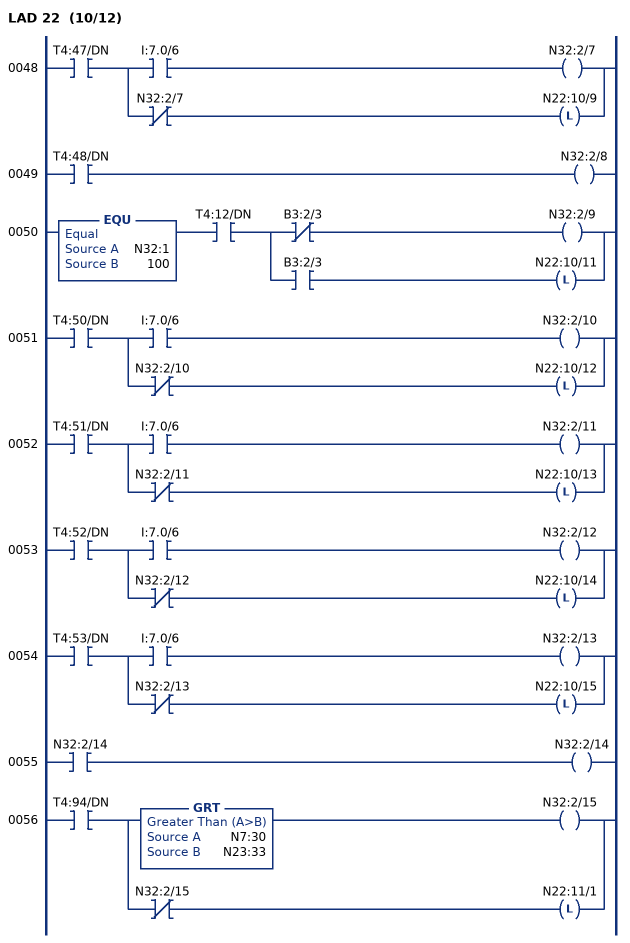
% Rung: 48 %
SOR XIC T4:47/DN BST XIC I:7.0/6 OTE N32:2/7 NXB XIO N32:2/7 OTL N22:10/9 BND EOR
% Rung: 49 %
SOR XIC T4:48/DN OTE N32:2/8 EOR
% Rung: 50 %
SOR EQU N32:1 100 XIC T4:12/DN BST XIO B3:2/3 OTE N32:2/9 NXB XIC B3:2/3 OTL N22:10/11 BND EOR
% Rung: 51 %
SOR XIC T4:50/DN BST XIC I:7.0/6 OTE N32:2/10 NXB XIO N32:2/10 OTL N22:10/12 BND EOR
% Rung: 52 %
SOR XIC T4:51/DN BST XIC I:7.0/6 OTE N32:2/11 NXB XIO N32:2/11 OTL N22:10/13 BND EOR
% Rung: 53 %
SOR XIC T4:52/DN BST XIC I:7.0/6 OTE N32:2/12 NXB XIO N32:2/12 OTL N22:10/14 BND EOR
% Rung: 54 %
SOR XIC T4:53/DN BST XIC I:7.0/6 OTE N32:2/13 NXB XIO N32:2/13 OTL N22:10/15 BND EOR
% Rung: 55 %
SOR XIC N32:2/14 OTE N32:2/14 EOR
% Rung: 56 %
SOR XIC T4:94/DN BST GRT N7:30 N23:33 OTE N32:2/15 NXB XIO N32:2/15 OTL N22:11/1 BND EOR

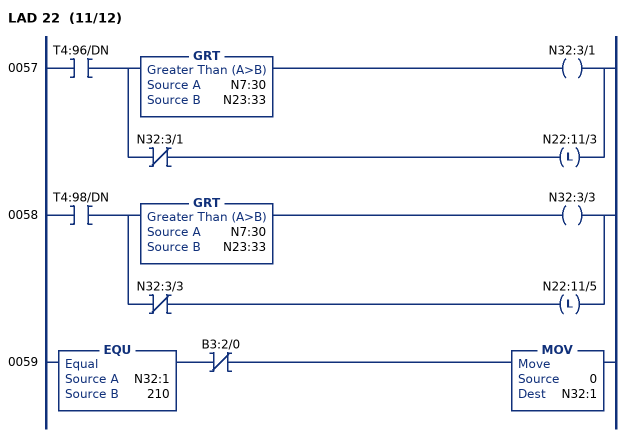
% Rung: 57 %
SOR XIC T4:96/DN BST GRT N7:30 N23:33 OTE N32:3/1 NXB XIO N32:3/1 OTL N22:11/3 BND EOR
% Rung: 58 %
SOR XIC T4:98/DN BST GRT N7:30 N23:33 OTE N32:3/3 NXB XIO N32:3/3 OTL N22:11/5 BND EOR
% Rung: 59 %
SOR EQU N32:1 210 XIO B3:2/0 MOV 0 N32:1 EOR

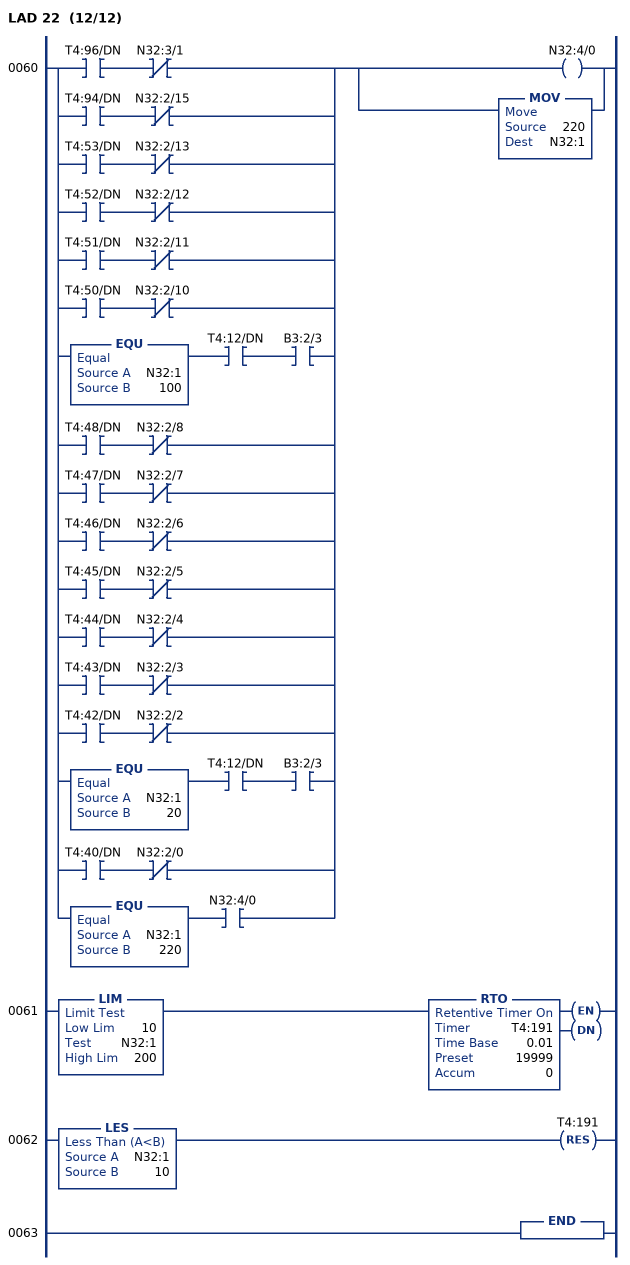
% Rung: 60 %
SOR BST XIC T4:96/DN XIO N32:3/1 NXB XIC T4:94/DN XIO N32:2/15 NXB XIC T4:53/DN XIO N32:2/13 NXB XIC T4:52/DN XIO N32:2/12 NXB XIC T4:51/DN XIO N32:2/11 NXB XIC T4:50/DN XIO N32:2/10 NXB EQU N32:1 100 XIC T4:12/DN XIC B3:2/3 NXB XIC T4:48/DN XIO N32:2/8 NXB XIC T4:47/DN XIO N32:2/7 NXB XIC T4:46/DN XIO N32:2/6 NXB XIC T4:45/DN XIO N32:2/5 NXB XIC T4:44/DN XIO N32:2/4 NXB XIC T4:43/DN XIO N32:2/3 NXB XIC T4:42/DN XIO N32:2/2 NXB EQU N32:1 20 XIC T4:12/DN XIC B3:2/3 NXB XIC T4:40/DN XIO N32:2/0 NXB EQU N32:1 220 XIC N32:4/0 BND BST OTE N32:4/0 NXB MOV 220 N32:1 BND EOR
% Rung: 61 %
SOR LIM 10 N32:1 200 RTO T4:191 0.01 19999 0 EOR
% Rung: 62 %
SOR LES N32:1 10 RES T4:191 EOR
% Rung: 63 %
SOR END EOR

LADDER 23
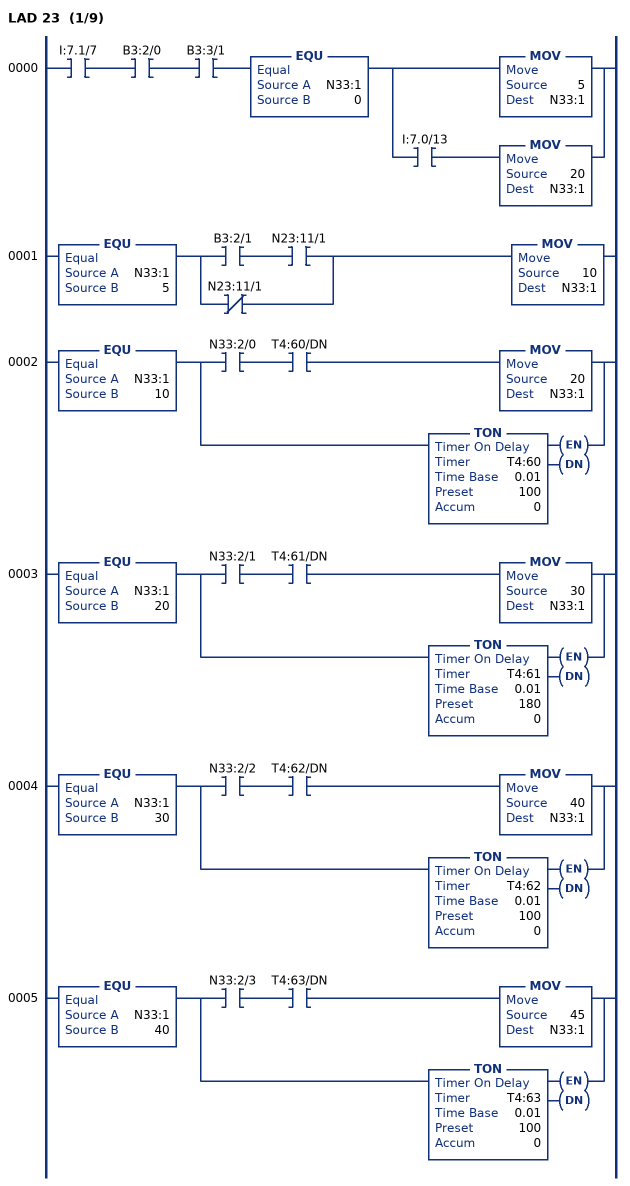
% Rung: 0 %
SOR XIC I:7.1/7 XIC B3:2/0 XIC B3:3/1 EQU N33:1 0 BST MOV 5 N33:1 NXB XIC I:7.0/13 MOV 20 N33:1 BND EOR
% Rung: 1 %
SOR EQU N33:1 5 BST XIC B3:2/1 XIC N23:11/1 NXB XIO N23:11/1 BND MOV 10 N33:1 EOR
% Rung: 2 %
SOR EQU N33:1 10 BST XIC N33:2/0 XIC T4:60/DN MOV 20 N33:1 NXB TON T4:60 0.01 100 0 BND EOR
% Rung: 3 %
SOR EQU N33:1 20 BST XIC N33:2/1 XIC T4:61/DN MOV 30 N33:1 NXB TON T4:61 0.01 180 0 BND EOR
% Rung: 4 %
SOR EQU N33:1 30 BST XIC N33:2/2 XIC T4:62/DN MOV 40 N33:1 NXB TON T4:62 0.01 100 0 BND EOR
% Rung: 5 %
SOR EQU N33:1 40 BST XIC N33:2/3 XIC T4:63/DN MOV 45 N33:1 NXB TON T4:63 0.01 100 0 BND EOR

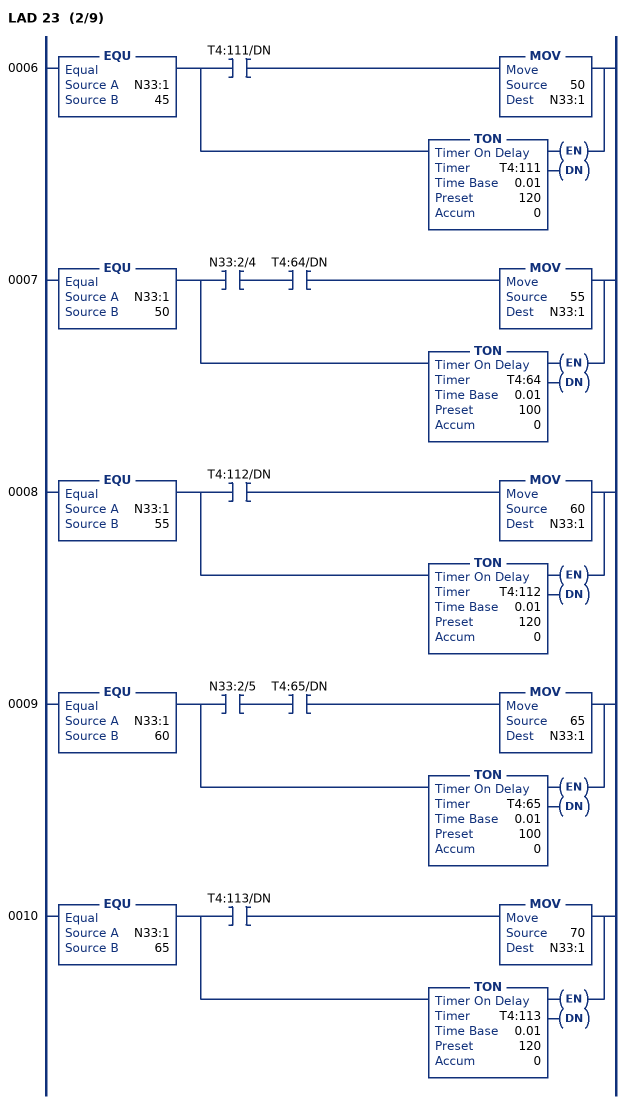
% Rung: 6 %
SOR EQU N33:1 45 BST XIC T4:111/DN MOV 50 N33:1 NXB TON T4:111 0.01 120 0 BND EOR
% Rung: 7 %
SOR EQU N33:1 50 BST XIC N33:2/4 XIC T4:64/DN MOV 55 N33:1 NXB TON T4:64 0.01 100 0 BND EOR
% Rung: 8 %
SOR EQU N33:1 55 BST XIC T4:112/DN MOV 60 N33:1 NXB TON T4:112 0.01 120 0 BND EOR
% Rung: 9 %
SOR EQU N33:1 60 BST XIC N33:2/5 XIC T4:65/DN MOV 65 N33:1 NXB TON T4:65 0.01 100 0 BND EOR
% Rung: 10 %
SOR EQU N33:1 65 BST XIC T4:113/DN MOV 70 N33:1 NXB TON T4:113 0.01 120 0 BND EOR

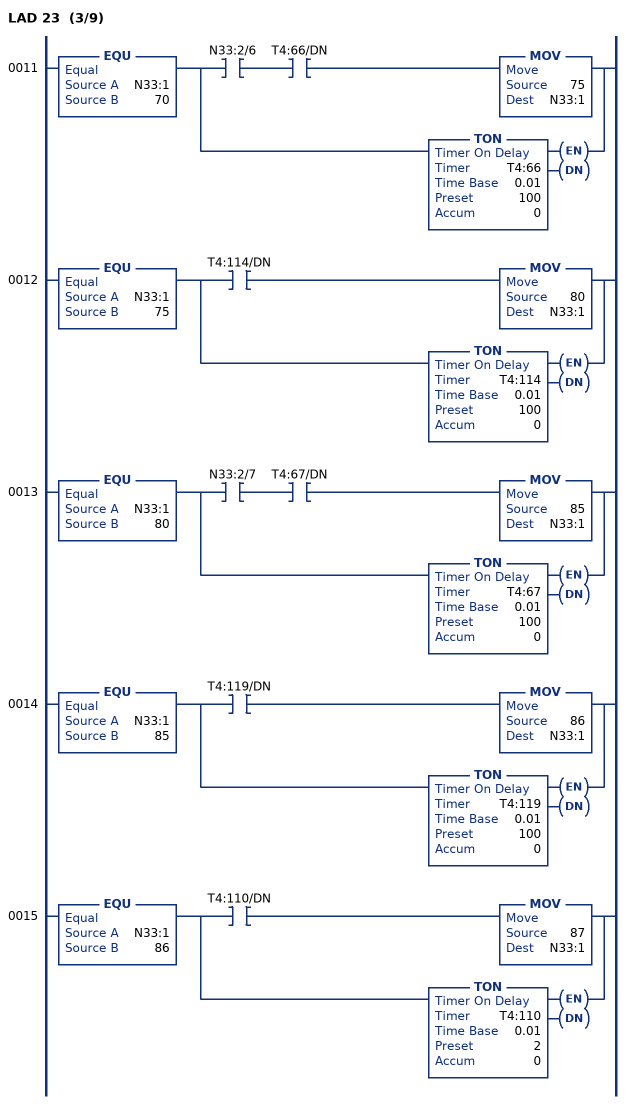
% Rung: 11 %
SOR EQU N33:1 70 BST XIC N33:2/6 XIC T4:66/DN MOV 75 N33:1 NXB TON T4:66 0.01 100 0 BND EOR
% Rung: 12 %
SOR EQU N33:1 75 BST XIC T4:114/DN MOV 80 N33:1 NXB TON T4:114 0.01 100 0 BND EOR
% Rung: 13 %
SOR EQU N33:1 80 BST XIC N33:2/7 XIC T4:67/DN MOV 85 N33:1 NXB TON T4:67 0.01 100 0 BND EOR
% Rung: 14 %
SOR EQU N33:1 85 BST XIC T4:119/DN MOV 86 N33:1 NXB TON T4:119 0.01 100 0 BND EOR
% Rung: 15 %
SOR EQU N33:1 86 BST XIC T4:110/DN MOV 87 N33:1 NXB TON T4:110 0.01 2 0 BND EOR

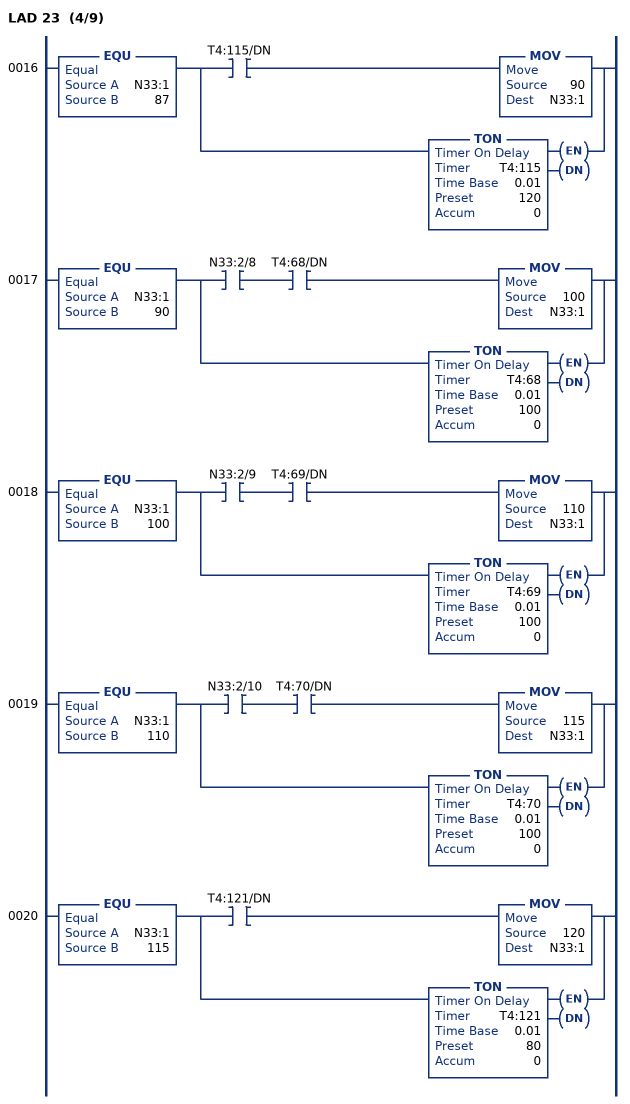
% Rung: 16 %
SOR EQU N33:1 87 BST XIC T4:115/DN MOV 90 N33:1 NXB TON T4:115 0.01 120 0 BND EOR
% Rung: 17 %
SOR EQU N33:1 90 BST XIC N33:2/8 XIC T4:68/DN MOV 100 N33:1 NXB TON T4:68 0.01 100 0 BND EOR
% Rung: 18 %
SOR EQU N33:1 100 BST XIC N33:2/9 XIC T4:69/DN MOV 110 N33:1 NXB TON T4:69 0.01 100 0 BND EOR
% Rung: 19 %
SOR EQU N33:1 110 BST XIC N33:2/10 XIC T4:70/DN MOV 115 N33:1 NXB TON T4:70 0.01 100 0 BND EOR
% Rung: 20 %
SOR EQU N33:1 115 BST XIC T4:121/DN MOV 120 N33:1 NXB TON T4:121 0.01 80 0 BND EOR

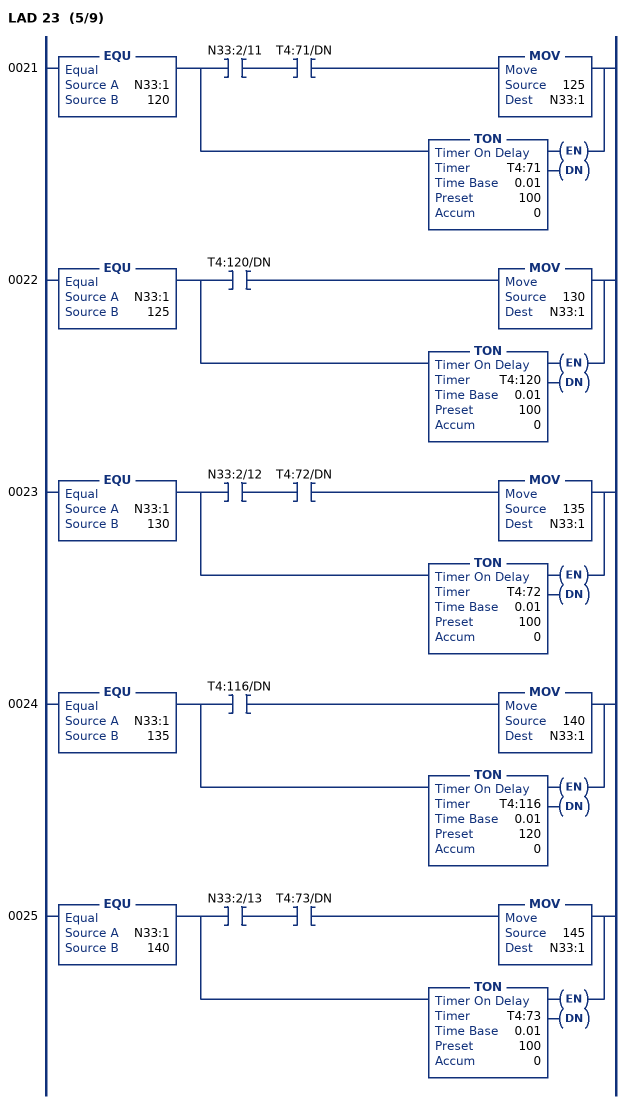
% Rung: 21 %
SOR EQU N33:1 120 BST XIC N33:2/11 XIC T4:71/DN MOV 125 N33:1 NXB TON T4:71 0.01 100 0 BND EOR
% Rung: 22 %
SOR EQU N33:1 125 BST XIC T4:120/DN MOV 130 N33:1 NXB TON T4:120 0.01 100 0 BND EOR
% Rung: 23 %
SOR EQU N33:1 130 BST XIC N33:2/12 XIC T4:72/DN MOV 135 N33:1 NXB TON T4:72 0.01 100 0 BND EOR
% Rung: 24 %
SOR EQU N33:1 135 BST XIC T4:116/DN MOV 140 N33:1 NXB TON T4:116 0.01 120 0 BND EOR
% Rung: 25 %
SOR EQU N33:1 140 BST XIC N33:2/13 XIC T4:73/DN MOV 145 N33:1 NXB TON T4:73 0.01 100 0 BND EOR

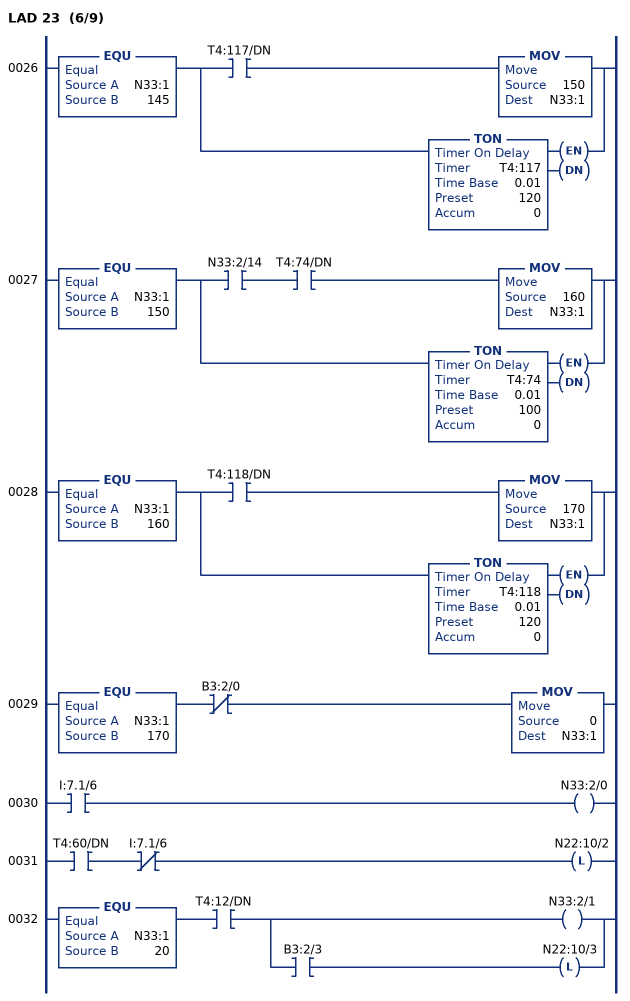
% Rung: 26 %
SOR EQU N33:1 145 BST XIC T4:117/DN MOV 150 N33:1 NXB TON T4:117 0.01 120 0 BND EOR
% Rung: 27 %
SOR EQU N33:1 150 BST XIC N33:2/14 XIC T4:74/DN MOV 160 N33:1 NXB TON T4:74 0.01 100 0 BND EOR
% Rung: 28 %
SOR EQU N33:1 160 BST XIC T4:118/DN MOV 170 N33:1 NXB TON T4:118 0.01 120 0 BND EOR
% Rung: 29 %
SOR EQU N33:1 170 XIO B3:2/0 MOV 0 N33:1 EOR
% Rung: 30 %
SOR XIC I:7.1/6 OTE N33:2/0 EOR
% Rung: 31 %
SOR XIC T4:60/DN XIO I:7.1/6 OTL N22:10/2 EOR
% Rung: 32 %
SOR EQU N33:1 20 XIC T4:12/DN BST OTE N33:2/1 NXB XIC B3:2/3 OTL N22:10/3 BND EOR

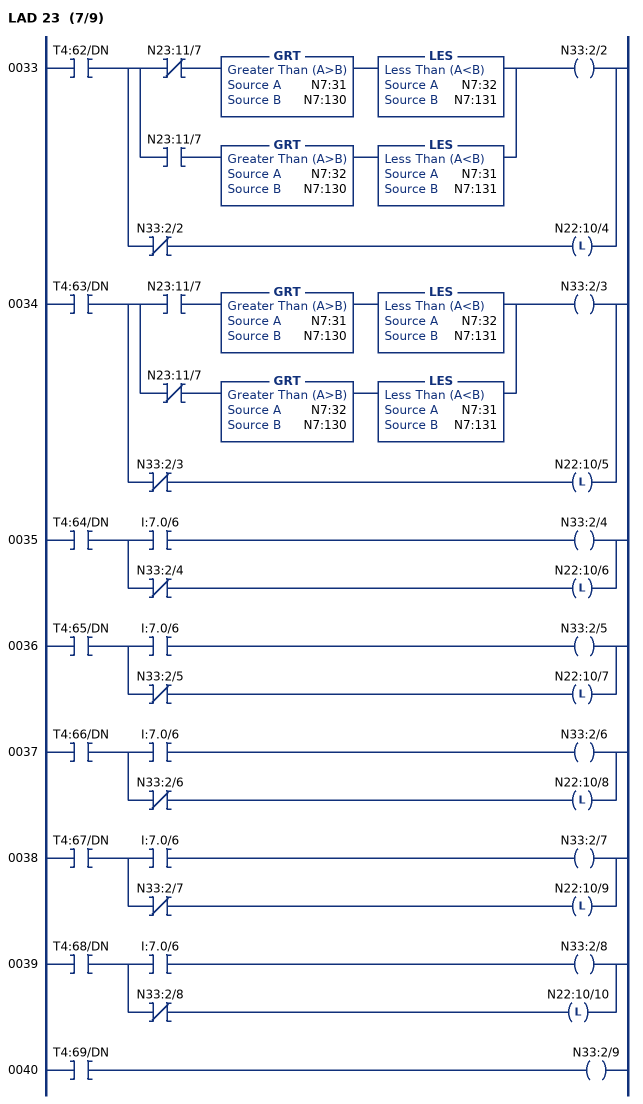
% Rung: 33 %
SOR XIC T4:62/DN BST BST XIO N23:11/7 GRT N7:31 N7:130 LES N7:32 N7:131 NXB XIC N23:11/7 GRT N7:32 N7:130 LES N7:31 N7:131 BND OTE N33:2/2 NXB XIO N33:2/2 OTL N22:10/4 BND EOR
% Rung: 34 %
SOR XIC T4:63/DN BST BST XIC N23:11/7 GRT N7:31 N7:130 LES N7:32 N7:131 NXB XIO N23:11/7 GRT N7:32 N7:130 LES N7:31 N7:131 BND OTE N33:2/3 NXB XIO N33:2/3 OTL N22:10/5 BND EOR
% Rung: 35 %
SOR XIC T4:64/DN BST XIC I:7.0/6 OTE N33:2/4 NXB XIO N33:2/4 OTL N22:10/6 BND EOR
% Rung: 36 %
SOR XIC T4:65/DN BST XIC I:7.0/6 OTE N33:2/5 NXB XIO N33:2/5 OTL N22:10/7 BND EOR
% Rung: 37 %
SOR XIC T4:66/DN BST XIC I:7.0/6 OTE N33:2/6 NXB XIO N33:2/6 OTL N22:10/8 BND EOR
% Rung: 38 %
SOR XIC T4:67/DN BST XIC I:7.0/6 OTE N33:2/7 NXB XIO N33:2/7 OTL N22:10/9 BND EOR
% Rung: 39 %
SOR XIC T4:68/DN BST XIC I:7.0/6 OTE N33:2/8 NXB XIO N33:2/8 OTL N22:10/10 BND EOR
% Rung: 40 %
SOR XIC T4:69/DN OTE N33:2/9 EOR

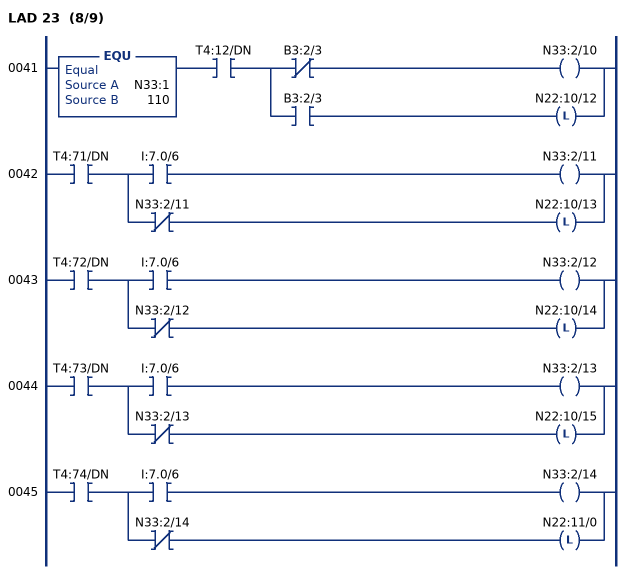
% Rung: 41 %
SOR EQU N33:1 110 XIC T4:12/DN BST XIO B3:2/3 OTE N33:2/10 NXB XIC B3:2/3 OTL N22:10/12 BND EOR
% Rung: 42 %
SOR XIC T4:71/DN BST XIC I:7.0/6 OTE N33:2/11 NXB XIO N33:2/11 OTL N22:10/13 BND EOR
% Rung: 43 %
SOR XIC T4:72/DN BST XIC I:7.0/6 OTE N33:2/12 NXB XIO N33:2/12 OTL N22:10/14 BND EOR
% Rung: 44 %
SOR XIC T4:73/DN BST XIC I:7.0/6 OTE N33:2/13 NXB XIO N33:2/13 OTL N22:10/15 BND EOR
% Rung: 45 %
SOR XIC T4:74/DN BST XIC I:7.0/6 OTE N33:2/14 NXB XIO N33:2/14 OTL N22:11/0 BND EOR

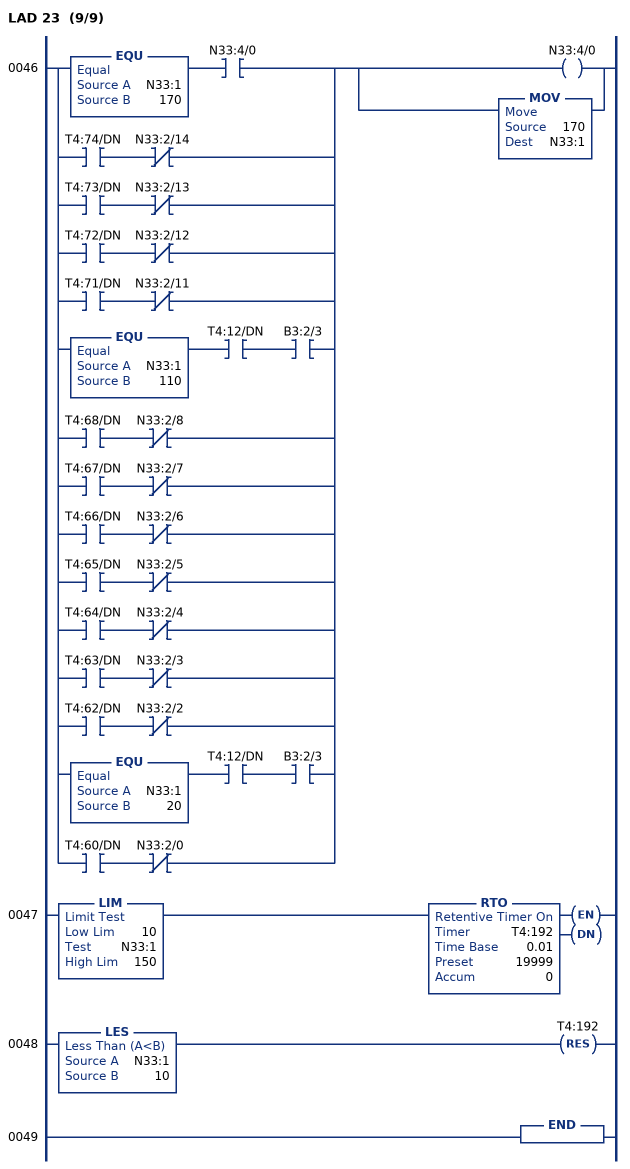
% Rung: 46 %
SOR BST EQU N33:1 170 XIC N33:4/0 NXB XIC T4:74/DN XIO N33:2/14 NXB XIC T4:73/DN XIO N33:2/13 NXB XIC T4:72/DN XIO N33:2/12 NXB XIC T4:71/DN XIO N33:2/11 NXB EQU N33:1 110 XIC T4:12/DN XIC B3:2/3 NXB XIC T4:68/DN XIO N33:2/8 NXB XIC T4:67/DN XIO N33:2/7 NXB XIC T4:66/DN XIO N33:2/6 NXB XIC T4:65/DN XIO N33:2/5 NXB XIC T4:64/DN XIO N33:2/4 NXB XIC T4:63/DN XIO N33:2/3 NXB XIC T4:62/DN XIO N33:2/2 NXB EQU N33:1 20 XIC T4:12/DN XIC B3:2/3 NXB XIC T4:60/DN XIO N33:2/0 BND BST OTE N33:4/0 NXB MOV 170 N33:1 BND EOR
% Rung: 47 %
SOR LIM 10 N33:1 150 RTO T4:192 0.01 19999 0 EOR
% Rung: 48 %
SOR LES N33:1 10 RES T4:192 EOR
% Rung: 49 %
SOR END EOR

LADDER 24
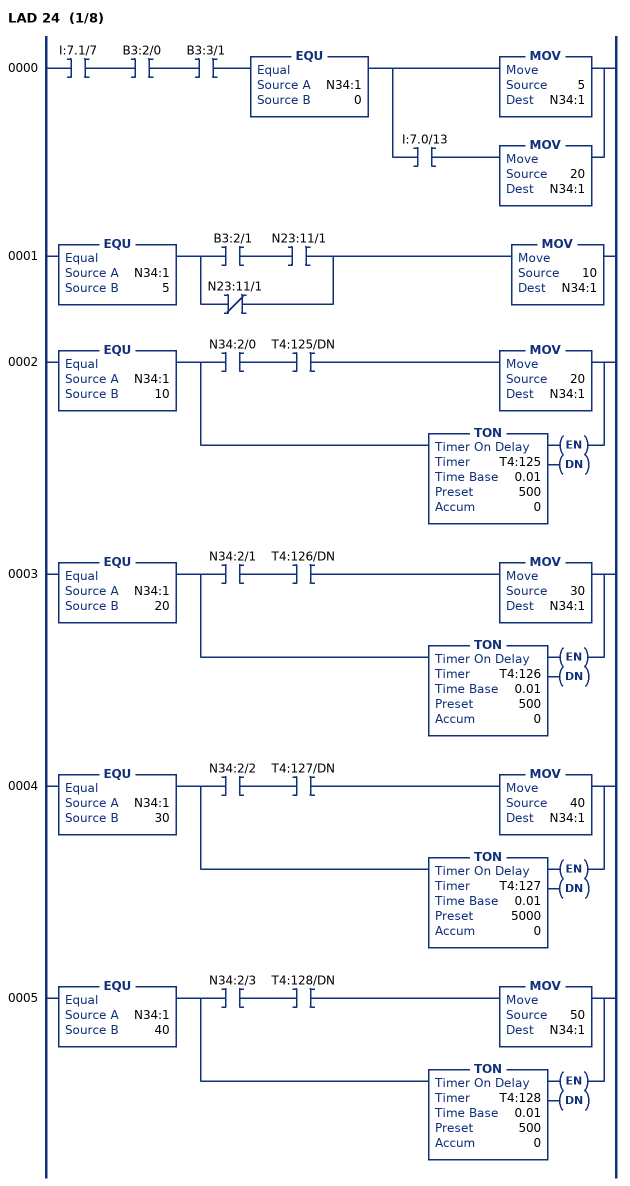
% Rung: 0 %
SOR XIC I:7.1/7 XIC B3:2/0 XIC B3:3/1 EQU N34:1 0 BST MOV 5 N34:1 NXB XIC I:7.0/13 MOV 20 N34:1 BND EOR
% Rung: 1 %
SOR EQU N34:1 5 BST XIC B3:2/1 XIC N23:11/1 NXB XIO N23:11/1 BND MOV 10 N34:1 EOR
% Rung: 2 %
SOR EQU N34:1 10 BST XIC N34:2/0 XIC T4:125/DN MOV 20 N34:1 NXB TON T4:125 0.01 500 0 BND EOR
% Rung: 3 %
SOR EQU N34:1 20 BST XIC N34:2/1 XIC T4:126/DN MOV 30 N34:1 NXB TON T4:126 0.01 500 0 BND EOR
% Rung: 4 %
SOR EQU N34:1 30 BST XIC N34:2/2 XIC T4:127/DN MOV 40 N34:1 NXB TON T4:127 0.01 5000 0 BND EOR
% Rung: 5 %
SOR EQU N34:1 40 BST XIC N34:2/3 XIC T4:128/DN MOV 50 N34:1 NXB TON T4:128 0.01 500 0 BND EOR

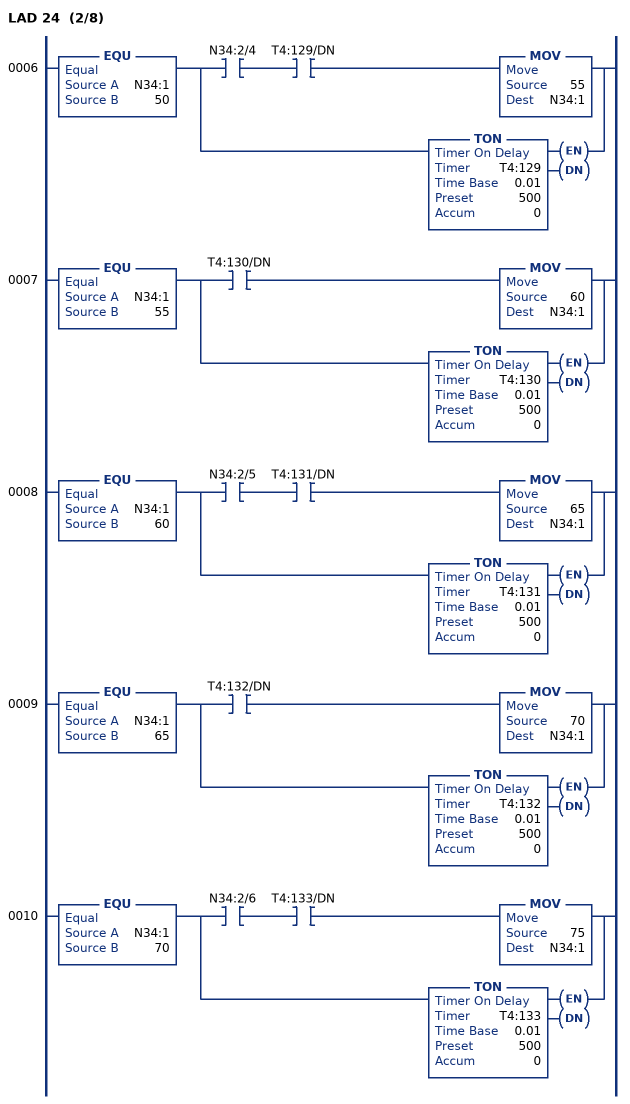
% Rung: 6 %
SOR EQU N34:1 50 BST XIC N34:2/4 XIC T4:129/DN MOV 55 N34:1 NXB TON T4:129 0.01 500 0 BND EOR
% Rung: 7 %
SOR EQU N34:1 55 BST XIC T4:130/DN MOV 60 N34:1 NXB TON T4:130 0.01 500 0 BND EOR
% Rung: 8 %
SOR EQU N34:1 60 BST XIC N34:2/5 XIC T4:131/DN MOV 65 N34:1 NXB TON T4:131 0.01 500 0 BND EOR
% Rung: 9 %
SOR EQU N34:1 65 BST XIC T4:132/DN MOV 70 N34:1 NXB TON T4:132 0.01 500 0 BND EOR
% Rung: 10 %
SOR EQU N34:1 70 BST XIC N34:2/6 XIC T4:133/DN MOV 75 N34:1 NXB TON T4:133 0.01 500 0 BND EOR

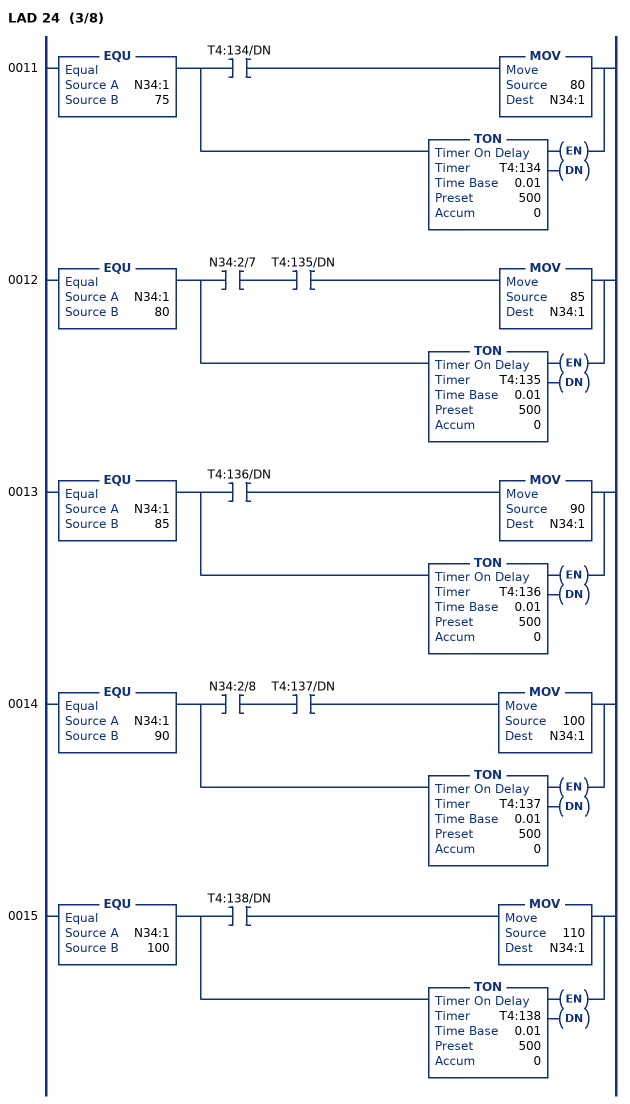
% Rung: 11 %
SOR EQU N34:1 75 BST XIC T4:134/DN MOV 80 N34:1 NXB TON T4:134 0.01 500 0 BND EOR
% Rung: 12 %
SOR EQU N34:1 80 BST XIC N34:2/7 XIC T4:135/DN MOV 85 N34:1 NXB TON T4:135 0.01 500 0 BND EOR
% Rung: 13 %
SOR EQU N34:1 85 BST XIC T4:136/DN MOV 90 N34:1 NXB TON T4:136 0.01 500 0 BND EOR
% Rung: 14 %
SOR EQU N34:1 90 BST XIC N34:2/8 XIC T4:137/DN MOV 100 N34:1 NXB TON T4:137 0.01 500 0 BND EOR
% Rung: 15 %
SOR EQU N34:1 100 BST XIC T4:138/DN MOV 110 N34:1 NXB TON T4:138 0.01 500 0 BND EOR

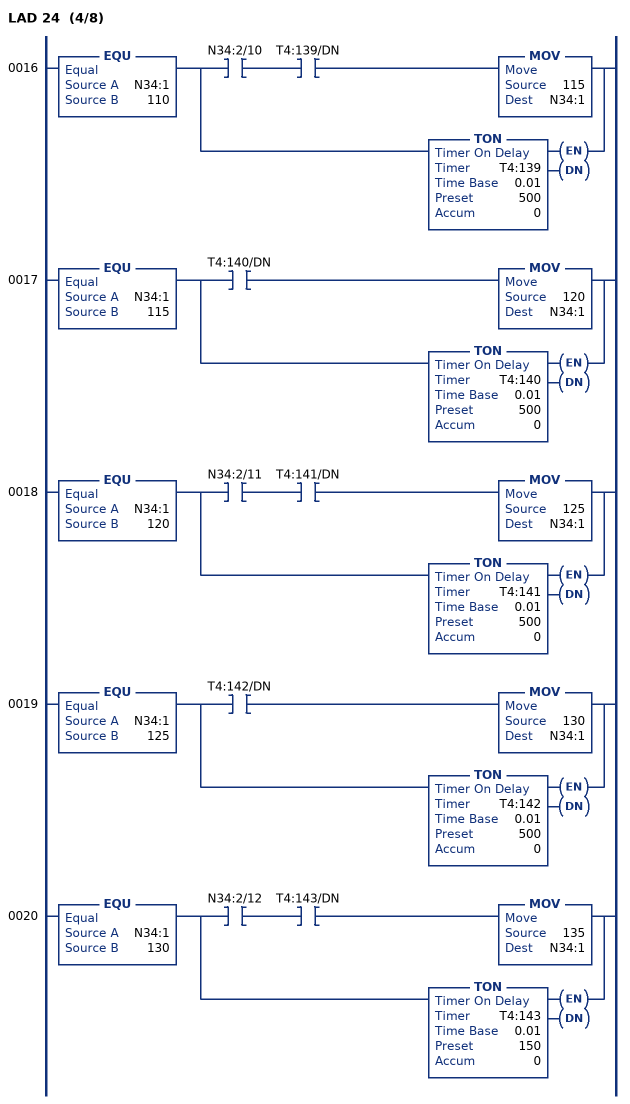
% Rung: 16 %
SOR EQU N34:1 110 BST XIC N34:2/10 XIC T4:139/DN MOV 115 N34:1 NXB TON T4:139 0.01 500 0 BND EOR
% Rung: 17 %
SOR EQU N34:1 115 BST XIC T4:140/DN MOV 120 N34:1 NXB TON T4:140 0.01 500 0 BND EOR
% Rung: 18 %
SOR EQU N34:1 120 BST XIC N34:2/11 XIC T4:141/DN MOV 125 N34:1 NXB TON T4:141 0.01 500 0 BND EOR
% Rung: 19 %
SOR EQU N34:1 125 BST XIC T4:142/DN MOV 130 N34:1 NXB TON T4:142 0.01 500 0 BND EOR
% Rung: 20 %
SOR EQU N34:1 130 BST XIC N34:2/12 XIC T4:143/DN MOV 135 N34:1 NXB TON T4:143 0.01 150 0 BND EOR

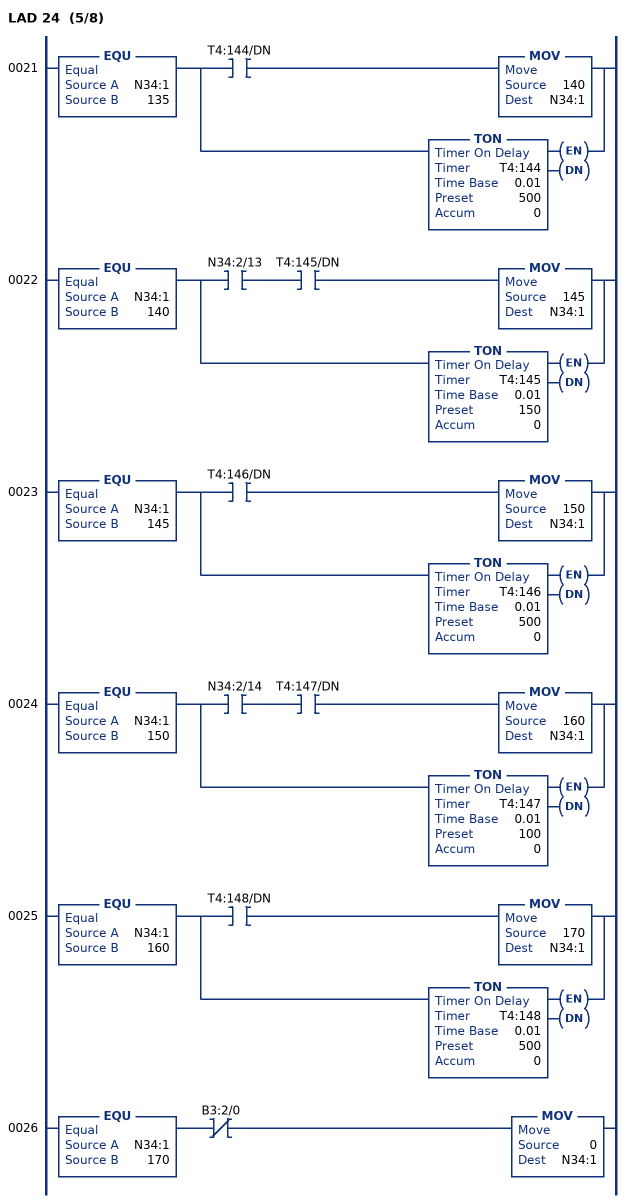
% Rung: 21 %
SOR EQU N34:1 135 BST XIC T4:144/DN MOV 140 N34:1 NXB TON T4:144 0.01 500 0 BND EOR
% Rung: 22 %
SOR EQU N34:1 140 BST XIC N34:2/13 XIC T4:145/DN MOV 145 N34:1 NXB TON T4:145 0.01 150 0 BND EOR
% Rung: 23 %
SOR EQU N34:1 145 BST XIC T4:146/DN MOV 150 N34:1 NXB TON T4:146 0.01 500 0 BND EOR
% Rung: 24 %
SOR EQU N34:1 150 BST XIC N34:2/14 XIC T4:147/DN MOV 160 N34:1 NXB TON T4:147 0.01 100 0 BND EOR
% Rung: 25 %
SOR EQU N34:1 160 BST XIC T4:148/DN MOV 170 N34:1 NXB TON T4:148 0.01 500 0 BND EOR
% Rung: 26 %
SOR EQU N34:1 170 XIO B3:2/0 MOV 0 N34:1 EOR

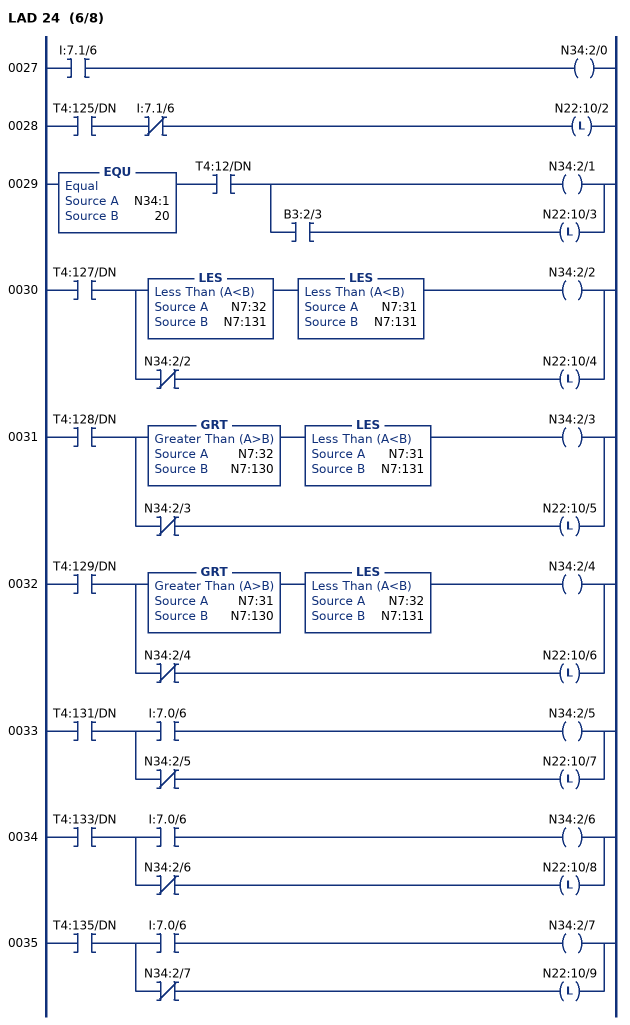
% Rung: 27 %
SOR XIC I:7.1/6 OTE N34:2/0 EOR
% Rung: 28 %
SOR XIC T4:125/DN XIO I:7.1/6 OTL N22:10/2 EOR
% Rung: 29 %
SOR EQU N34:1 20 XIC T4:12/DN BST OTE N34:2/1 NXB XIC B3:2/3 OTL N22:10/3 BND EOR
% Rung: 30 %
SOR XIC T4:127/DN BST LES N7:32 N7:131 LES N7:31 N7:131 OTE N34:2/2 NXB XIO N34:2/2 OTL N22:10/4 BND EOR
% Rung: 31 %
SOR XIC T4:128/DN BST GRT N7:32 N7:130 LES N7:31 N7:131 OTE N34:2/3 NXB XIO N34:2/3 OTL N22:10/5 BND EOR
% Rung: 32 %
SOR XIC T4:129/DN BST GRT N7:31 N7:130 LES N7:32 N7:131 OTE N34:2/4 NXB XIO N34:2/4 OTL N22:10/6 BND EOR
% Rung: 33 %
SOR XIC T4:131/DN BST XIC I:7.0/6 OTE N34:2/5 NXB XIO N34:2/5 OTL N22:10/7 BND EOR
% Rung: 34 %
SOR XIC T4:133/DN BST XIC I:7.0/6 OTE N34:2/6 NXB XIO N34:2/6 OTL N22:10/8 BND EOR
% Rung: 35 %
SOR XIC T4:135/DN BST XIC I:7.0/6 OTE N34:2/7 NXB XIO N34:2/7 OTL N22:10/9 BND EOR

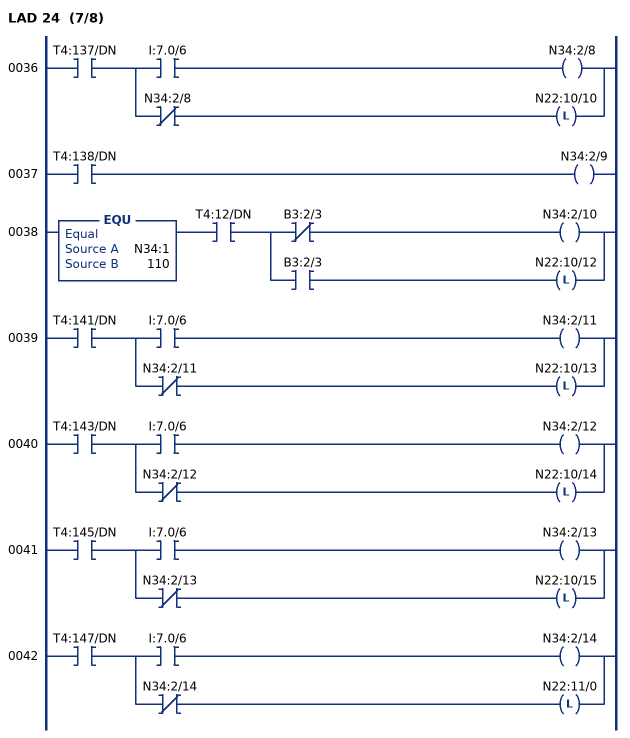
% Rung: 36 %
SOR XIC T4:137/DN BST XIC I:7.0/6 OTE N34:2/8 NXB XIO N34:2/8 OTL N22:10/10 BND EOR
% Rung: 37 %
SOR XIC T4:138/DN OTE N34:2/9 EOR
% Rung: 38 %
SOR EQU N34:1 110 XIC T4:12/DN BST XIO B3:2/3 OTE N34:2/10 NXB XIC B3:2/3 OTL N22:10/12 BND EOR
% Rung: 39 %
SOR XIC T4:141/DN BST XIC I:7.0/6 OTE N34:2/11 NXB XIO N34:2/11 OTL N22:10/13 BND EOR
% Rung: 40 %
SOR XIC T4:143/DN BST XIC I:7.0/6 OTE N34:2/12 NXB XIO N34:2/12 OTL N22:10/14 BND EOR
% Rung: 41 %
SOR XIC T4:145/DN BST XIC I:7.0/6 OTE N34:2/13 NXB XIO N34:2/13 OTL N22:10/15 BND EOR
% Rung: 42 %
SOR XIC T4:147/DN BST XIC I:7.0/6 OTE N34:2/14 NXB XIO N34:2/14 OTL N22:11/0 BND EOR

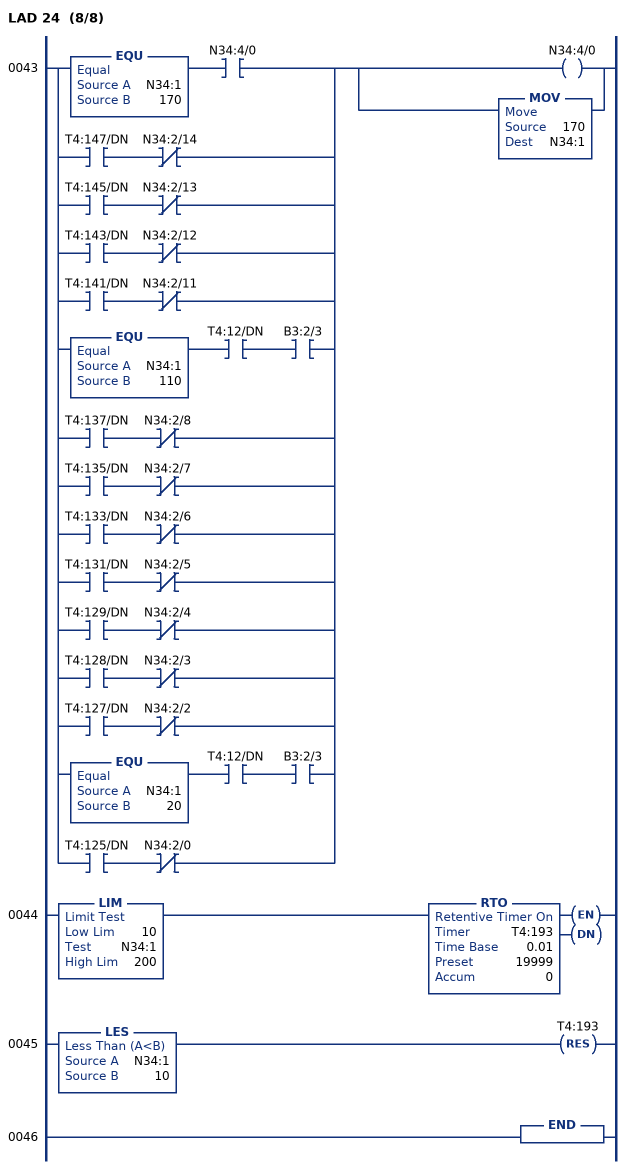
% Rung: 43 %
SOR BST EQU N34:1 170 XIC N34:4/0 NXB XIC T4:147/DN XIO N34:2/14 NXB XIC T4:145/DN XIO N34:2/13 NXB XIC T4:143/DN XIO N34:2/12 NXB XIC T4:141/DN XIO N34:2/11 NXB EQU N34:1 110 XIC T4:12/DN XIC B3:2/3 NXB XIC T4:137/DN XIO N34:2/8 NXB XIC T4:135/DN XIO N34:2/7 NXB XIC T4:133/DN XIO N34:2/6 NXB XIC T4:131/DN XIO N34:2/5 NXB XIC T4:129/DN XIO N34:2/4 NXB XIC T4:128/DN XIO N34:2/3 NXB XIC T4:127/DN XIO N34:2/2 NXB EQU N34:1 20 XIC T4:12/DN XIC B3:2/3 NXB XIC T4:125/DN XIO N34:2/0 BND BST OTE N34:4/0 NXB MOV 170 N34:1 BND EOR
% Rung: 44 %
SOR LIM 10 N34:1 200 RTO T4:193 0.01 19999 0 EOR
% Rung: 45 %
SOR LES N34:1 10 RES T4:193 EOR
% Rung: 46 %
SOR END EOR

DATA TABLE (non-zero values as saved)
DATA B3
% B3:0 % 0X8003 0X0005 0X0002 0X0001 0X0000 0X0000 0X0000 0X0000 0X0000 0X0000
DATA T4
% .PRE .ACC %
% T4:0 % 3 1
% T4:1 % 2 0
% T4:2 % 10 0
% T4:3 % 2 0
% T4:4 % 50 0
% T4:5 % 50 0
% T4:6 % 2 2
% T4:7 % 1 1
% T4:8 % 20 20
% T4:9 % 100 100
% T4:10 % 50 0
% T4:11 % 50 0
% T4:12 % 150 0
% T4:13 % 167 0
% T4:14 % 166 0
% T4:15 % 50 50
% T4:16 % 60 0
% T4:17 % 90 0
% T4:18 % 170 0
% T4:19 % 30 30
% T4:20 % 100 0
% T4:21 % 100 0
% T4:22 % 50 0
% T4:23 % 100 0
% T4:24 % 150 0
% T4:25 % 150 0
% T4:26 % 100 0
% T4:27 % 150 0
% T4:28 % 30 0
% T4:29 % 100 0
% T4:30 % 150 0
% T4:31 % 150 0
% T4:32 % 100 0
% T4:33 % 350 0
% T4:34 % 100 0
% T4:35 % 350 0
% T4:36 % 150 0
% T4:37 % 150 0
% T4:38 % 100 0
% T4:39 % 50 0
% T4:40 % 100 0
% T4:41 % 20 0
% T4:42 % 90 0
% T4:43 % 90 0
% T4:44 % 150 0
% T4:45 % 150 0
% T4:46 % 150 0
% T4:47 % 150 0
% T4:48 % 20 0
% T4:49 % 70 0
% T4:50 % 150 0
% T4:51 % 150 0
% T4:52 % 150 0
% T4:53 % 150 0
% T4:54 % 100 0
% T4:55 % 10 0
% T4:56 % 70 0
% T4:57 % 70 0
% T4:58 % 110 0
% T4:59 % 110 0
% T4:60 % 100 0
% T4:61 % 180 0
% T4:62 % 100 0
% T4:63 % 100 0
% T4:64 % 100 0
% T4:65 % 100 0
% T4:66 % 100 0
% T4:67 % 100 0
% T4:68 % 100 0
% T4:69 % 100 0
% T4:70 % 100 0
% T4:71 % 100 0
% T4:72 % 100 0
% T4:73 % 100 0
% T4:74 % 100 0
% T4:75 % 100 0
% T4:76 % 200 0
% T4:77 % 100 0
% T4:78 % 50 0
% T4:80 % 60 0
% T4:81 % 60 0
% T4:82 % 60 0
% T4:83 % 60 0
% T4:84 % 60 0
% T4:85 % 60 0
% T4:86 % 60 0
% T4:87 % 60 0
% T4:88 % 60 0
% T4:89 % 100 0
% T4:90 % 80 0
% T4:91 % 50 0
% T4:92 % 50 0
% T4:93 % 100 0
% T4:94 % 500 0
% T4:95 % 500 0
% T4:96 % 500 0
% T4:97 % 600 0
% T4:98 % 500 0
% T4:99 % 200 0
% T4:100 % 200 0
% T4:101 % 200 0
% T4:102 % 200 0
% T4:103 % 100 0
% T4:104 % 100 0
% T4:105 % 120 0
% T4:106 % 120 0
% T4:107 % 120 0
% T4:108 % 120 0
% T4:109 % 120 0
% T4:110 % 2 0
% T4:111 % 120 0
% T4:112 % 120 0
% T4:113 % 120 0
% T4:114 % 100 0
% T4:115 % 120 0
% T4:116 % 120 0
% T4:117 % 120 0
% T4:118 % 120 0
% T4:119 % 100 0
% T4:120 % 100 0
% T4:121 % 80 0
% T4:125 % 500 0
% T4:126 % 500 0
% T4:127 % 5000 0
% T4:128 % 500 0
% T4:129 % 500 0
% T4:130 % 500 0
% T4:131 % 500 0
% T4:132 % 500 0
% T4:133 % 500 0
% T4:134 % 500 0
% T4:135 % 500 0
% T4:136 % 500 0
% T4:137 % 500 0
% T4:138 % 500 0
% T4:139 % 500 0
% T4:140 % 500 0
% T4:141 % 500 0
% T4:142 % 500 0
% T4:143 % 150 0
% T4:144 % 500 0
% T4:145 % 150 0
% T4:146 % 500 0
% T4:147 % 100 0
% T4:148 % 500 0
% T4:190 % 19999 0
% T4:191 % 19999 0
% T4:192 % 19999 0
% T4:193 % 19999 0
% T4:199 % 150 0
DATA N7
% N7:0 % 30 102 0 0 200 400 1870 0 0 0
% N7:10 % 30 102 0 0 200 400 1870 0 0 0
% N7:20 % 0 76 0 0 0 0 0 1870 102 30
% N7:30 % -50 -25 -25 0 0 0 0 0 0 0
% N7:50 % 0 1 1 0 0 0 0 0 0 0
% N7:60 % 10 2 102 0 0 0 0 0 0 0
% N7:80 % 2 75 150 5 167 333 0 0 0 0
% N7:90 % 0 0 0 0 0 0 0 0 1 3
% N7:100 % 1 0 0 80 0 0 0 0 0 0
% N7:110 % 20 20 15 0 0 82 10 0 0 0
% N7:130 % 68 12 0 0 0 0 0 0 0 0
DATA F8
% F8:0 % 0 102 1 0 0
% F8:5 % 0.85 0.15 0.5 0.5 3
DATA ST20
% ST20:0 % ".01\0A\0D"
% ST20:1 % "1"
% ST20:2 % "10.21\0A\0D"
% ST20:3 % "2"
% ST20:5 % "0\0A"
% ST20:10 % "."
DATA N21
% N21:10 % 195 130 1 408 384 300 2 16 1 80
% N21:20 % 0 10 0 0 15 20 0 0 1 15
% N21:30 % 30 917 50 0 0 0 0 0 0 0
DATA N22
% N22:10 % 0 0 4 1 -25 -25 0 0 0 0
% N22:20 % 3740 204 10 -50 917 3 0 0 0 0
DATA N23
% N23:10 % 195 130 1 204 192 30 2 16 1 80
% N23:20 % 0 10 0 0 15 20 0 0 1 15
% N23:30 % 30 917 50 0 0 0 0 0 0 0
DATA N31
% N31:0 % 1 0 0 79 0 0 79 0 0 0
% N31:10 % 18 0 0 0 0 0 0 0 0 0
DATA N32
% N32:0 % 1 0 0 69 0 0 0 0 0 0
% N32:10 % 22 0 0 0 0 0 0 0 0 0
DATA N33
% N33:0 % 1 0 0 0 0 0 0 0 0 0
% N33:10 % 17 0 0 0 0 0 0 0 0 0
DATA N34
% N34:0 % 1 0 0 0 0 0 0 0 0 0
% N34:10 % 3 0 0 0 0 0 0 0 0 0
DATA N40
% N40:0 % 230 2690 1345 0 0 0 0 0 0 0
DATA N41
% N41:0 % 230 2690 120 1 1 -1225 0 0 0 0
% N41:10 % 3
DATA N50
% N50:0 % 30 102 1870 0 101 103 29 31 0 0
DATA N51
% N51:0 % 1 102 0 0 0 0 0 0 0 0
% N51:10 % 4 0 0 0 0 0 0 0 0 0
